// TIA Portal V16 export
// export: Created 2022-11-14T17:35:22.8319203Z, ExportSetting WithDefaults, DisplayName Totally Integrated Automation Portal, DisplayVersion V16, DisplayName TIA Portal Version Control Interface, DisplayVersion V16, DisplayName TIA Portal Openness, DisplayVersion V16, DisplayName STEP 7 Professional, DisplayVersion V16, DisplayName STEP 7 Safety, DisplayVersion V16, DisplayName WinCC Advanced, DisplayVersion V16
FUNCTION "Inverter_CW_Assembly" : Void   // FC16, FBD
{ S7_Optimized_Access := 'TRUE' }
VERSION : 0.1
// stored: AutoNumber false, IsIECCheckEnabled false, SetENOAutomatically false, UDAEnableTagReadback false
   VAR_INPUT
      CW_Off1_On : Bool;
      CW_Off2 : Bool;
      CW_Off3 : Bool;
      CW_enable_operation : Bool;
      CW_no_lock_RFG : Bool;
      CW_no_stop_RFG : Bool;
      CW_enable_setpoint : Bool;
      CW_acknowledge : Bool;
      CW_not_used_1 : Bool;
      CW_not_used_2 : Bool;
      CW_PLC_is_Master : Bool;
      CW_direction_reversal : Bool;
      CW_not_used_3 : Bool;
      CW_motortpoti_up : Bool;
      CW_motortpoti_down : Bool;
      CW_not_used_4 : Bool;
   END_VAR
   VAR_IN_OUT
      Control_word : Word;
   END_VAR
BEGIN

REGION Network 1
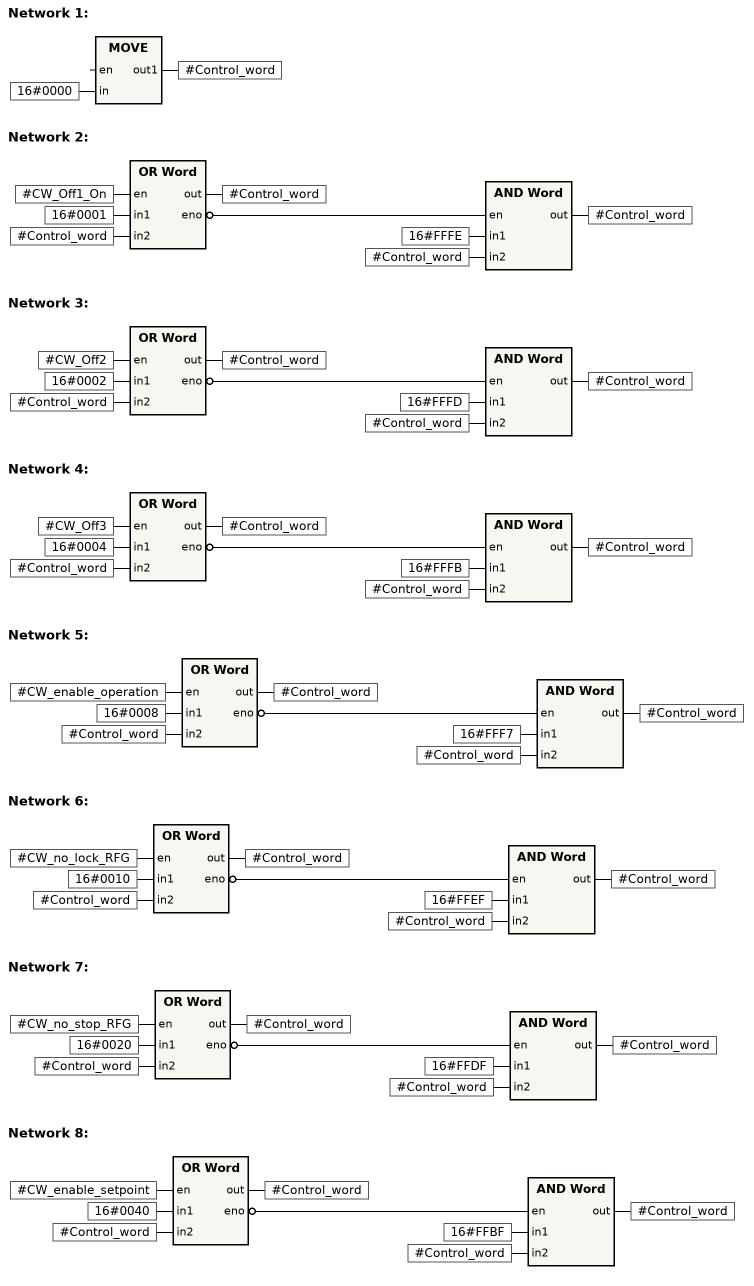
   #Control_word := 16#0000;
END_REGION

REGION Network 2
   IF #CW_Off1_On THEN #Control_word := 16#0001 OR #Control_word; END_IF;
   IF NOT #CW_Off1_On THEN #Control_word := 16#FFFE AND #Control_word; END_IF;
END_REGION

REGION Network 3
   IF #CW_Off2 THEN #Control_word := 16#0002 OR #Control_word; END_IF;
   IF NOT #CW_Off2 THEN #Control_word := 16#FFFD AND #Control_word; END_IF;
END_REGION

REGION Network 4
   IF #CW_Off3 THEN #Control_word := 16#0004 OR #Control_word; END_IF;
   IF NOT #CW_Off3 THEN #Control_word := 16#FFFB AND #Control_word; END_IF;
END_REGION

REGION Network 5
   IF #CW_enable_operation THEN #Control_word := 16#0008 OR #Control_word; END_IF;
   IF NOT #CW_enable_operation THEN #Control_word := 16#FFF7 AND #Control_word; END_IF;
END_REGION

REGION Network 6
   IF #CW_no_lock_RFG THEN #Control_word := 16#0010 OR #Control_word; END_IF;
   IF NOT #CW_no_lock_RFG THEN #Control_word := 16#FFEF AND #Control_word; END_IF;
END_REGION

REGION Network 7
   IF #CW_no_stop_RFG THEN #Control_word := 16#0020 OR #Control_word; END_IF;
   IF NOT #CW_no_stop_RFG THEN #Control_word := 16#FFDF AND #Control_word; END_IF;
END_REGION

REGION Network 8
   IF #CW_enable_setpoint THEN #Control_word := 16#0040 OR #Control_word; END_IF;
   IF NOT #CW_enable_setpoint THEN #Control_word := 16#FFBF AND #Control_word; END_IF;
END_REGION

REGION Network 9
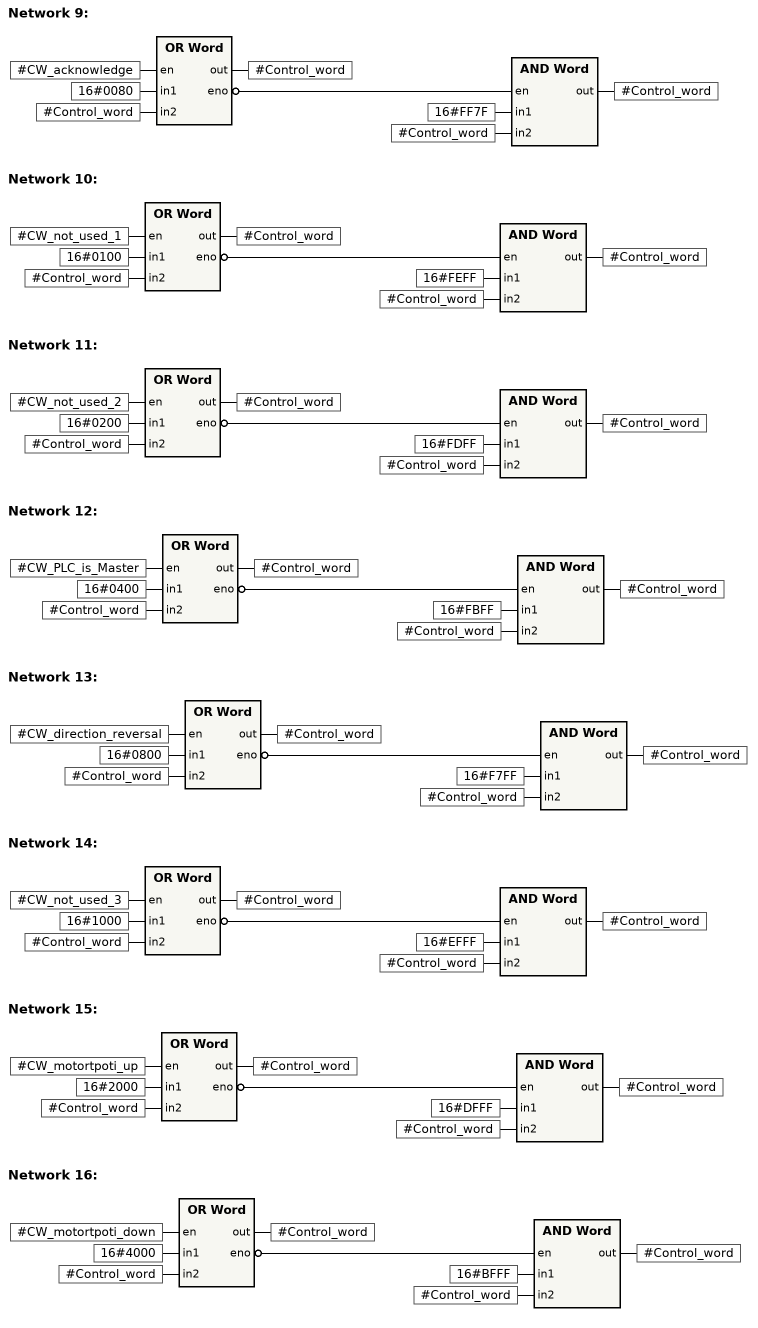
   IF #CW_acknowledge THEN #Control_word := 16#0080 OR #Control_word; END_IF;
   IF NOT #CW_acknowledge THEN #Control_word := 16#FF7F AND #Control_word; END_IF;
END_REGION

REGION Network 10
   IF #CW_not_used_1 THEN #Control_word := 16#0100 OR #Control_word; END_IF;
   IF NOT #CW_not_used_1 THEN #Control_word := 16#FEFF AND #Control_word; END_IF;
END_REGION

REGION Network 11
   IF #CW_not_used_2 THEN #Control_word := 16#0200 OR #Control_word; END_IF;
   IF NOT #CW_not_used_2 THEN #Control_word := 16#FDFF AND #Control_word; END_IF;
END_REGION

REGION Network 12
   IF #CW_PLC_is_Master THEN #Control_word := 16#0400 OR #Control_word; END_IF;
   IF NOT #CW_PLC_is_Master THEN #Control_word := 16#FBFF AND #Control_word; END_IF;
END_REGION

REGION Network 13
   IF #CW_direction_reversal THEN #Control_word := 16#0800 OR #Control_word; END_IF;
   IF NOT #CW_direction_reversal THEN #Control_word := 16#F7FF AND #Control_word; END_IF;
END_REGION

REGION Network 14
   IF #CW_not_used_3 THEN #Control_word := 16#1000 OR #Control_word; END_IF;
   IF NOT #CW_not_used_3 THEN #Control_word := 16#EFFF AND #Control_word; END_IF;
END_REGION

REGION Network 15
   IF #CW_motortpoti_up THEN #Control_word := 16#2000 OR #Control_word; END_IF;
   IF NOT #CW_motortpoti_up THEN #Control_word := 16#DFFF AND #Control_word; END_IF;
END_REGION

REGION Network 16
   IF #CW_motortpoti_down THEN #Control_word := 16#4000 OR #Control_word; END_IF;
   IF NOT #CW_motortpoti_down THEN #Control_word := 16#BFFF AND #Control_word; END_IF;
END_REGION

REGION Network 17
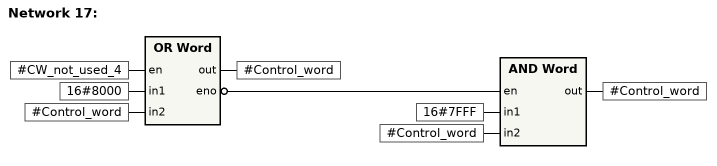
   IF #CW_not_used_4 THEN #Control_word := 16#8000 OR #Control_word; END_IF;
   IF NOT #CW_not_used_4 THEN #Control_word := 16#7FFF AND #Control_word; END_IF;
END_REGION
END_FUNCTION
